RoboDK station: KR10.rdk

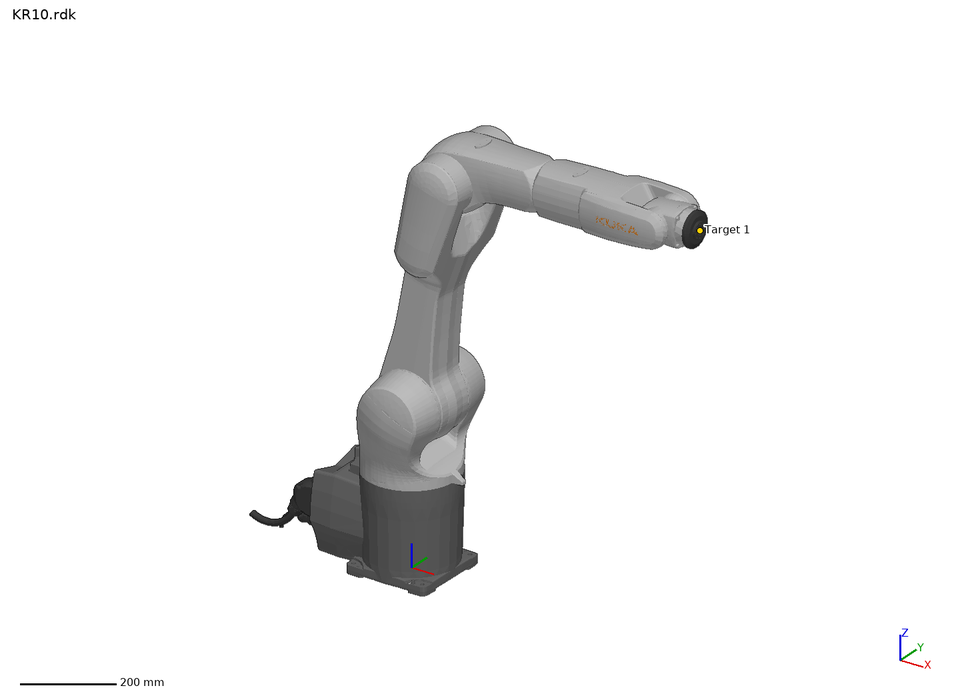
[picture v0: the station drawn from its stored meshes, robots at their saved joint values, targets as dots, program paths as lines]
Station KR10 (saved by RoboDK 5.6.8). Poses are relative to the parent item; angles as X-Y-Z fixed-axis rotations.
  - frame KUKA KR 10 R1100-2 Base at (0, 0, 0) mm
    - robot KUKA KR 10 R1100-2: 6 axes, payload 10.9 kg, reach 1101 mm, repeatability 0.02 mm, weight 56.5 kg
        modified DH rows (alpha deg, a mm, theta deg, d mm): 0, 0, 0, 400; -90, 25, 0, 0; 0, 560, -90, 0; -90, 25, 0, 515; 90, 0, 0, 0; -90, 0, 180, 90
        joint limits [-170, -190, -120, -185, -120, -350] to [170, 45, 156, 185, 120, 350]; home [0, -90, 90, 0, 0, 0]; saved at [0, -79.383, 78.316, 0, 1.067, 0]
    - target Target 1 (Cartesian target) at (732.62, 0, 985) mm, rotated rx 0 ry 90 rz 0 deg; joints [0, -79.383, 78.316, 0, 1.067, 0] of KUKA KR 10 R1100-2
